ABB RobotStudio station: LAB2_def.rspag

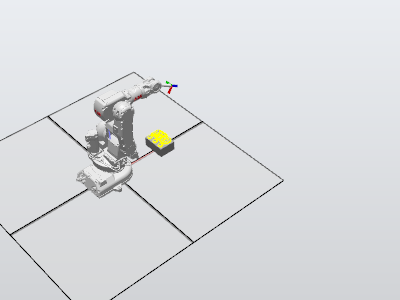
--- station ---
Station LAB2_def (saved by RobotStudio 25.1.11167.1)
Controller IRB140_6_81
  mechanical unit ROB_1: IRB140_6_81_C_03, 6 joints, base frame (0, 0, 0) mm
Layout (positions relative to the parent item):
  - IRB140_6_81_C_03 [mechanism, from %ABB.RobotStudio.Models.IRB140%\IRB140_6_81_C_G_03.rslib] at (0, 0, 0) mm; joint values [0, 0, 0, 0, 0.5236, 0] (rad or m)
  - Herramienta [mechanism, from Components\Herramienta.rslib] at (506.29, 0, 679.5) mm, rotated rx 180 ry 60 rz 180 deg
  - Pastel_MD [part] at (500, 0, 0) mm, rotated rx 0 ry 0 rz -90 deg, size 210.2 x 150 x 100 mm
  - Frame_4 [frame] at (-0.01, 0.2, 170.9) mm
Attachment: Herramienta is attached to IRB140_6_81_C_03 / Link6
Targets, tools, work objects and paths stored in the station and not in the controller backup, written as RAPID:
! task T_ROB1
MODULE Module1
  CONST robtarget Target_710:=[[91.512,-90.324660702,-494.059660254],[0.612372436,0.353553391,-0.353553391,0.612372436],[0,-1,0,0],[9E+09,9E+09,9E+09,9E+09,9E+09,9E+09]];
ENDMODULE


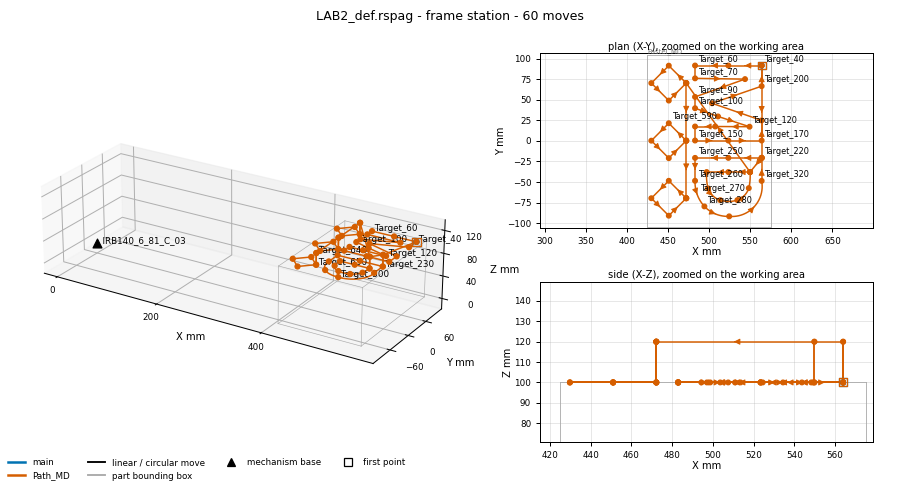
[picture p0: tool path of LAB2_def.rspag in frame station, 60 of 60 moves have a stored position in this frame; points joined in program order, loops and branches not executed]
--- Controller Data/IRB140_6_81/RAPID/TASK1/PROGMOD/CalibData.mod ---
MODULE CalibData
    PERS tooldata tHerramienta:=[TRUE,[[-0.01,0.197,170.898],[1,0,0,0]],[0.7,[0,0,1],[1,0,0,0],0,0,0]];
    TASK PERS wobjdata WObj_MD:=[FALSE,TRUE,"",[[0,0,0],[1,0,0,0]],[[563.974,91.709,100],[0,-0.707106781,0.707106781,0]]];
ENDMODULE

--- Controller Data/IRB140_6_81/RAPID/TASK1/PROGMOD/Module1.mod ---
MODULE Module1
        CONST robtarget Target_40:=[[0,0,0],[0.707106781,0,0,0.707106781],[0,0,0,0],[9E+09,9E+09,9E+09,9E+09,9E+09,9E+09]];
    CONST robtarget Target_50:=[[0,40.5,0],[0.707106781,0,0,0.707106781],[0,0,0,0],[9E+09,9E+09,9E+09,9E+09,9E+09,9E+09]];
    CONST robtarget Target_60:=[[0,81,0],[0.707106781,0,0,0.707106781],[0,0,0,0],[9E+09,9E+09,9E+09,9E+09,9E+09,9E+09]];
    CONST robtarget Target_70:=[[15.583,81,0],[0.707106781,0,0,0.707106781],[0,0,0,0],[9E+09,9E+09,9E+09,9E+09,9E+09,9E+09]];
    CONST robtarget Target_80:=[[16.52,20.243,0],[0.707106781,0,0,0.707106781],[0,0,0,0],[9E+09,9E+09,9E+09,9E+09,9E+09,9E+09]];
    CONST robtarget Target_90:=[[38.173,81,0],[0.707106781,0,0,0.707106781],[0,0,0,0],[9E+09,9E+09,9E+09,9E+09,9E+09,9E+09]];
    CONST robtarget Target_100:=[[51.925,81,0],[0.707106781,0,0,0.707106781],[0,0,0,0],[9E+09,9E+09,9E+09,9E+09,9E+09,9E+09]];
    CONST robtarget Target_110:=[[61.913,53.076,0],[0.707106781,0,0,0.707106781],[0,0,0,0],[9E+09,9E+09,9E+09,9E+09,9E+09,9E+09]];
    CONST robtarget Target_120:=[[74.411,14.746,0],[0.707106781,0,0,0.707106781],[0,0,0,0],[9E+09,9E+09,9E+09,9E+09,9E+09,9E+09]];
    CONST robtarget Target_130:=[[74.149,56.423,0],[0.707106781,0,0,0.707106781],[0,0,0,0],[9E+09,9E+09,9E+09,9E+09,9E+09,9E+09]];
    CONST robtarget Target_140:=[[74.149,81,0],[0.707106781,0,0,0.707106781],[0,0,0,0],[9E+09,9E+09,9E+09,9E+09,9E+09,9E+09]];
    CONST robtarget Target_150:=[[91.197,81,0],[0.707106781,0,0,0.707106781],[0,0,0,0],[9E+09,9E+09,9E+09,9E+09,9E+09,9E+09]];
    CONST robtarget Target_160:=[[91.197,40.5,0],[0.707106781,0,0,0.707106781],[0,0,0,0],[9E+09,9E+09,9E+09,9E+09,9E+09,9E+09]];
    CONST robtarget Target_170:=[[91.197,0,0],[0.707106781,0,0,0.707106781],[0,0,0,0],[9E+09,9E+09,9E+09,9E+09,9E+09,9E+09]];
    CONST robtarget Target_180:=[[66.776,0,0],[0.707106781,0,0,0.707106781],[0,0,0,0],[9E+09,9E+09,9E+09,9E+09,9E+09,9E+09]];
    CONST robtarget Target_190:=[[45.912,60.344,0],[0.707106781,0,0,0.707106781],[0,0,0,0],[9E+09,9E+09,9E+09,9E+09,9E+09,9E+09]];
    CONST robtarget Target_200:=[[25.1,0,0],[0.707106781,0,0,0.707106781],[0,0,0,0],[9E+09,9E+09,9E+09,9E+09,9E+09,9E+09]];
    CONST robtarget Target_210:=[[0,0,0],[0.707106781,0,0,0.707106781],[0,0,0,0],[9E+09,9E+09,9E+09,9E+09,9E+09,9E+09]];
    CONST robtarget Target_220:=[[112.302,0,-20],[0.707106781,0,0,0.707106781],[0,0,0,0],[9E+09,9E+09,9E+09,9E+09,9E+09,9E+09]];
    CONST robtarget Target_230:=[[112.302,0,0],[0.707106781,0,0,0.707106781],[0,0,0,0],[9E+09,9E+09,9E+09,9E+09,9E+09,9E+09]];
    CONST robtarget Target_240:=[[112.302,40.5,0],[0.707106781,0,0,0.707106781],[0,0,0,0],[9E+09,9E+09,9E+09,9E+09,9E+09,9E+09]];
    CONST robtarget Target_250:=[[112.302,81,0],[0.707106781,0,0,0.707106781],[0,0,0,0],[9E+09,9E+09,9E+09,9E+09,9E+09,9E+09]];
    CONST robtarget Target_260:=[[140.173,81,0],[0.707106781,0,0,0.707106781],[0,0,0,0],[9E+09,9E+09,9E+09,9E+09,9E+09,9E+09]];
    CONST robtarget Target_270:=[[156.902,78.38,0],[0.707106781,0,0,0.707106781],[0,0,0,0],[9E+09,9E+09,9E+09,9E+09,9E+09,9E+09]];
    CONST robtarget Target_280:=[[171.339,69.626,0],[0.707106781,0,0,0.707106781],[0,0,0,0],[9E+09,9E+09,9E+09,9E+09,9E+09,9E+09]];
    CONST robtarget Target_290:=[[180.612,55.877,0],[0.707106781,0,0,0.707106781],[0,0,0,0],[9E+09,9E+09,9E+09,9E+09,9E+09,9E+09]];
    CONST robtarget Target_300:=[[183.418,39.48,0],[0.707106781,0,0,0.707106781],[0,0,0,0],[9E+09,9E+09,9E+09,9E+09,9E+09,9E+09]];
    CONST robtarget Target_310:=[[171.876,9.164,0],[0.707106781,0,0,0.707106781],[0,0,0,0],[9E+09,9E+09,9E+09,9E+09,9E+09,9E+09]];
    CONST robtarget Target_320:=[[140.278,0,0],[0.707106781,0,0,0.707106781],[0,0,0,0],[9E+09,9E+09,9E+09,9E+09,9E+09,9E+09]];
    CONST robtarget Target_330:=[[112.302,0,0],[0.707106781,0,0,0.707106781],[0,0,0,0],[9E+09,9E+09,9E+09,9E+09,9E+09,9E+09]];
    CONST robtarget Target_340:=[[112.302,0,-20],[0.707106781,0,0,0.707106781],[0,0,0,0],[9E+09,9E+09,9E+09,9E+09,9E+09,9E+09]];
    CONST robtarget Target_350:=[[129.558,14.119,-20],[0.707106781,0,0,0.707106781],[0,0,0,0],[9E+09,9E+09,9E+09,9E+09,9E+09,9E+09]];
    CONST robtarget Target_360:=[[129.558,14.119,0],[0.707106781,0,0,0.707106781],[0,0,0,0],[9E+09,9E+09,9E+09,9E+09,9E+09,9E+09]];
    CONST robtarget Target_370:=[[129.558,40.5,0],[0.707106781,0,0,0.707106781],[0,0,0,0],[9E+09,9E+09,9E+09,9E+09,9E+09,9E+09]];
    CONST robtarget Target_380:=[[129.558,66.881,0],[0.707106781,0,0,0.707106781],[0,0,0,0],[9E+09,9E+09,9E+09,9E+09,9E+09,9E+09]];
    CONST robtarget Target_390:=[[138.97,66.881,0],[0.707106781,0,0,0.707106781],[0,0,0,0],[9E+09,9E+09,9E+09,9E+09,9E+09,9E+09]];
    CONST robtarget Target_400:=[[149.416,65.253,0],[0.707106781,0,0,0.707106781],[0,0,0,0],[9E+09,9E+09,9E+09,9E+09,9E+09,9E+09]];
    CONST robtarget Target_410:=[[158.266,59.56,0],[0.707106781,0,0,0.707106781],[0,0,0,0],[9E+09,9E+09,9E+09,9E+09,9E+09,9E+09]];
    CONST robtarget Target_420:=[[163.729,50.369,0],[0.707106781,0,0,0.707106781],[0,0,0,0],[9E+09,9E+09,9E+09,9E+09,9E+09,9E+09]];
    CONST robtarget Target_430:=[[165.273,39.741,0],[0.707106781,0,0,0.707106781],[0,0,0,0],[9E+09,9E+09,9E+09,9E+09,9E+09,9E+09]];
    CONST robtarget Target_440:=[[163.645,29.499,0],[0.707106781,0,0,0.707106781],[0,0,0,0],[9E+09,9E+09,9E+09,9E+09,9E+09,9E+09]];
    CONST robtarget Target_450:=[[157.952,20.89,0],[0.707106781,0,0,0.707106781],[0,0,0,0],[9E+09,9E+09,9E+09,9E+09,9E+09,9E+09]];
    CONST robtarget Target_460:=[[149.11,15.659,0],[0.707106781,0,0,0.707106781],[0,0,0,0],[9E+09,9E+09,9E+09,9E+09,9E+09,9E+09]];
    CONST robtarget Target_470:=[[138.918,14.119,0],[0.707106781,0,0,0.707106781],[0,0,0,0],[9E+09,9E+09,9E+09,9E+09,9E+09,9E+09]];
    CONST robtarget Target_480:=[[129.558,14.119,0],[0.707106781,0,0,0.707106781],[0,0,0,0],[9E+09,9E+09,9E+09,9E+09,9E+09,9E+09]];
    CONST robtarget Target_490:=[[129.558,14.119,-20],[0.707106781,0,0,0.707106781],[0,0,0,0],[9E+09,9E+09,9E+09,9E+09,9E+09,9E+09]];
    CONST robtarget Target_500:=[[21.391,91.731,-20],[0.707106781,0,0,0.707106781],[0,0,0,0],[9E+09,9E+09,9E+09,9E+09,9E+09,9E+09]];
    CONST robtarget Target_510:=[[21.391,91.731,0],[0.707106781,0,0,0.707106781],[0,0,0,0],[9E+09,9E+09,9E+09,9E+09,9E+09,9E+09]];
    CONST robtarget Target_520:=[[0.178,112.944,0],[0.707106781,0,0,0.707106781],[0,0,0,0],[9E+09,9E+09,9E+09,9E+09,9E+09,9E+09]];
    CONST robtarget Target_530:=[[21.391,134.157,0],[0.707106781,0,0,0.707106781],[0,0,0,0],[9E+09,9E+09,9E+09,9E+09,9E+09,9E+09]];
    CONST robtarget Target_540:=[[42.605,112.944,0],[0.707106781,0,0,0.707106781],[0,0,0,0],[9E+09,9E+09,9E+09,9E+09,9E+09,9E+09]];
    CONST robtarget Target_550:=[[21.391,91.731,0],[0.707106781,0,0,0.707106781],[0,0,0,0],[9E+09,9E+09,9E+09,9E+09,9E+09,9E+09]];
    CONST robtarget Target_560:=[[21.391,91.731,-20],[0.707106781,0,0,0.707106781],[0,0,0,0],[9E+09,9E+09,9E+09,9E+09,9E+09,9E+09]];
    CONST robtarget Target_570:=[[91.391,91.731,-20],[0.707106781,0,0,0.707106781],[0,0,0,0],[9E+09,9E+09,9E+09,9E+09,9E+09,9E+09]];
    CONST robtarget Target_580:=[[91.391,91.731,0],[0.707106781,0,0,0.707106781],[0,0,0,0],[9E+09,9E+09,9E+09,9E+09,9E+09,9E+09]];
    CONST robtarget Target_590:=[[70.178,112.944,0],[0.707106781,0,0,0.707106781],[0,0,0,0],[9E+09,9E+09,9E+09,9E+09,9E+09,9E+09]];
    CONST robtarget Target_600:=[[91.391,134.157,0],[0.707106781,0,0,0.707106781],[0,0,0,0],[9E+09,9E+09,9E+09,9E+09,9E+09,9E+09]];
    CONST robtarget Target_610:=[[112.605,112.944,0],[0.707106781,0,0,0.707106781],[0,0,0,0],[9E+09,9E+09,9E+09,9E+09,9E+09,9E+09]];
    CONST robtarget Target_620:=[[91.391,91.731,0],[0.707106781,0,0,0.707106781],[0,0,0,0],[9E+09,9E+09,9E+09,9E+09,9E+09,9E+09]];
    CONST robtarget Target_630:=[[91.391,91.731,-20],[0.707106781,0,0,0.707106781],[0,0,0,0],[9E+09,9E+09,9E+09,9E+09,9E+09,9E+09]];
    CONST robtarget Target_640:=[[161.391,91.731,-20],[0.707106781,0,0,0.707106781],[0,0,0,0],[9E+09,9E+09,9E+09,9E+09,9E+09,9E+09]];
    CONST robtarget Target_650:=[[161.391,91.731,0],[0.707106781,0,0,0.707106781],[0,0,0,0],[9E+09,9E+09,9E+09,9E+09,9E+09,9E+09]];
    CONST robtarget Target_660:=[[140.178,112.944,0],[0.707106781,0,0,0.707106781],[0,0,0,0],[9E+09,9E+09,9E+09,9E+09,9E+09,9E+09]];
    CONST robtarget Target_670:=[[161.391,134.157,0],[0.707106781,0,0,0.707106781],[0,0,0,0],[9E+09,9E+09,9E+09,9E+09,9E+09,9E+09]];
    CONST robtarget Target_680:=[[182.605,112.944,0],[0.707106781,0,0,0.707106781],[0,0,0,0],[9E+09,9E+09,9E+09,9E+09,9E+09,9E+09]];
    CONST robtarget Target_690:=[[161.391,91.731,0],[0.707106781,0,0,0.707106781],[0,0,0,0],[9E+09,9E+09,9E+09,9E+09,9E+09,9E+09]];
    CONST robtarget Target_700:=[[161.391,91.731,-20],[0.707106781,0,0,0.707106781],[0,0,0,0],[9E+09,9E+09,9E+09,9E+09,9E+09,9E+09]];
!***********************************************************
    !
    ! Module:  Module1
    !
    ! Description:
    !   <Insert description here>
    !
    ! Author: M_o-_
    !
    ! Version: 1.0
    !
    !***********************************************************


    !***********************************************************
    !
    ! Procedure main
    !
    !   This is the entry point of your program
    !
    !***********************************************************
    PROC main()
        MoveL Target_40,v100,fine,tHerramienta\WObj:=WObj_MD;
        !Path_MD;
    ENDPROC
    PROC Path_MD()
        MoveL Target_40,v100,fine,tHerramienta\WObj:=WObj_MD;
        MoveL Target_50,v50,z0,tHerramienta\WObj:=WObj_MD;
        MoveL Target_60,v50,z0,tHerramienta\WObj:=WObj_MD;
        MoveL Target_70,v50,z0,tHerramienta\WObj:=WObj_MD;
        MoveL Target_80,v50,z0,tHerramienta\WObj:=WObj_MD;
        MoveL Target_90,v50,z0,tHerramienta\WObj:=WObj_MD;
        MoveL Target_100,v50,z0,tHerramienta\WObj:=WObj_MD;
        MoveL Target_110,v50,z0,tHerramienta\WObj:=WObj_MD;
        MoveL Target_120,v50,z0,tHerramienta\WObj:=WObj_MD;
        MoveL Target_130,v50,z0,tHerramienta\WObj:=WObj_MD;
        MoveL Target_140,v50,z0,tHerramienta\WObj:=WObj_MD;
        MoveL Target_150,v50,z0,tHerramienta\WObj:=WObj_MD;
        MoveL Target_160,v50,z0,tHerramienta\WObj:=WObj_MD;
        MoveL Target_170,v50,z0,tHerramienta\WObj:=WObj_MD;
        MoveL Target_180,v50,z0,tHerramienta\WObj:=WObj_MD;
        MoveL Target_190,v50,z0,tHerramienta\WObj:=WObj_MD;
        MoveL Target_200,v50,z0,tHerramienta\WObj:=WObj_MD;
        MoveL Target_210,v50,z0,tHerramienta\WObj:=WObj_MD;
        MoveL Target_220,v300,z5,tHerramienta\WObj:=WObj_MD;
        MoveL Target_230,v100,fine,tHerramienta\WObj:=WObj_MD;
        MoveL Target_240,v50,z0,tHerramienta\WObj:=WObj_MD;
        MoveL Target_250,v50,z0,tHerramienta\WObj:=WObj_MD;
        MoveL Target_260,v50,z0,tHerramienta\WObj:=WObj_MD;
        MoveC Target_270,Target_280,v50,z0,tHerramienta\WObj:=WObj_MD;
        MoveC Target_290,Target_300,v50,z0,tHerramienta\WObj:=WObj_MD;
        MoveC Target_310,Target_320,v50,z0,tHerramienta\WObj:=WObj_MD;
        MoveL Target_330,v50,z0,tHerramienta\WObj:=WObj_MD;
        MoveL Target_340,v300,z5,tHerramienta\WObj:=WObj_MD;
        MoveL Target_350,v100,z5,tHerramienta\WObj:=WObj_MD;
        MoveL Target_360,v100,fine,tHerramienta\WObj:=WObj_MD;
        MoveL Target_370,v50,z0,tHerramienta\WObj:=WObj_MD;
        MoveL Target_380,v50,z0,tHerramienta\WObj:=WObj_MD;
        MoveC Target_390,Target_400,v50,z0,tHerramienta\WObj:=WObj_MD;
        MoveC Target_410,Target_420,v50,z0,tHerramienta\WObj:=WObj_MD;
        MoveC Target_430,Target_440,v50,z0,tHerramienta\WObj:=WObj_MD;
        MoveC Target_450,Target_460,v50,z0,tHerramienta\WObj:=WObj_MD;
        MoveC Target_470,Target_480,v50,z0,tHerramienta\WObj:=WObj_MD;
        MoveL Target_490,v100,z5,tHerramienta\WObj:=WObj_MD;
        MoveL Target_500,v300,z5,tHerramienta\WObj:=WObj_MD;
        MoveL Target_510,v100,fine,tHerramienta\WObj:=WObj_MD;
        MoveL Target_520,v50,z0,tHerramienta\WObj:=WObj_MD;
        MoveL Target_530,v50,z0,tHerramienta\WObj:=WObj_MD;
        MoveL Target_540,v50,z0,tHerramienta\WObj:=WObj_MD;
        MoveL Target_550,v50,z0,tHerramienta\WObj:=WObj_MD;
        MoveL Target_560,v100,z5,tHerramienta\WObj:=WObj_MD;
        MoveL Target_570,v300,z5,tHerramienta\WObj:=WObj_MD;
        MoveL Target_580,v100,fine,tHerramienta\WObj:=WObj_MD;
        MoveL Target_590,v50,z0,tHerramienta\WObj:=WObj_MD;
        MoveL Target_600,v50,z0,tHerramienta\WObj:=WObj_MD;
        MoveL Target_610,v50,z0,tHerramienta\WObj:=WObj_MD;
        MoveL Target_620,v50,z0,tHerramienta\WObj:=WObj_MD;
        MoveL Target_630,v100,z5,tHerramienta\WObj:=WObj_MD;
        MoveL Target_640,v300,z5,tHerramienta\WObj:=WObj_MD;
        MoveL Target_650,v100,fine,tHerramienta\WObj:=WObj_MD;
        MoveL Target_660,v50,z0,tHerramienta\WObj:=WObj_MD;
        MoveL Target_670,v50,z0,tHerramienta\WObj:=WObj_MD;
        MoveL Target_680,v50,z0,tHerramienta\WObj:=WObj_MD;
        MoveL Target_690,v50,z0,tHerramienta\WObj:=WObj_MD;
        MoveL Target_700,v300,z5,tHerramienta\WObj:=WObj_MD;
    ENDPROC
ENDMODULE
